FUNCTION_BLOCK SpecificFanPower
VAR_INPUT
END_VAR
VAR_OUTPUT
END_VAR
VAR
END_VAR

END_FUNCTION_BLOCK

(* stored: Version 1.1.0.1, ProductVersion 3.1.4024.3
   POU SpecificFanPower: Id {953b4b95-9e24-49ca-9799-05c35d71dc6f}, SpecialFunc None *)
